% RSLogix 500 project fast_test.RSS, saved by version 8.30.00.16 %
PROJECT "UNTITLED"    % processor: Bul.1763 MicroLogix 1100 Series A %

PROGRAM FILES
  LAD 2 "MAIN"  6 rungs
  LAD 3 "CIRC_FIFO"  10 rungs

DATA FILES
  O0 OUTPUT  4 elements
  I1 INPUT  6 elements
  S2 STATUS  66 elements
  B3 BINARY  1 elements
  T4 TIMER  1 elements
  C5 COUNTER  1 elements
  R6 CONTROL  1 elements
  N7 INTEGER  6 elements
  F8 FLOAT  1 elements
  N252 LINE0  32 elements
  N253 LINE 1  32 elements
  N254 LINE 2  32 elements
  N255 LINE3  32 elements

LADDER 2 "MAIN"
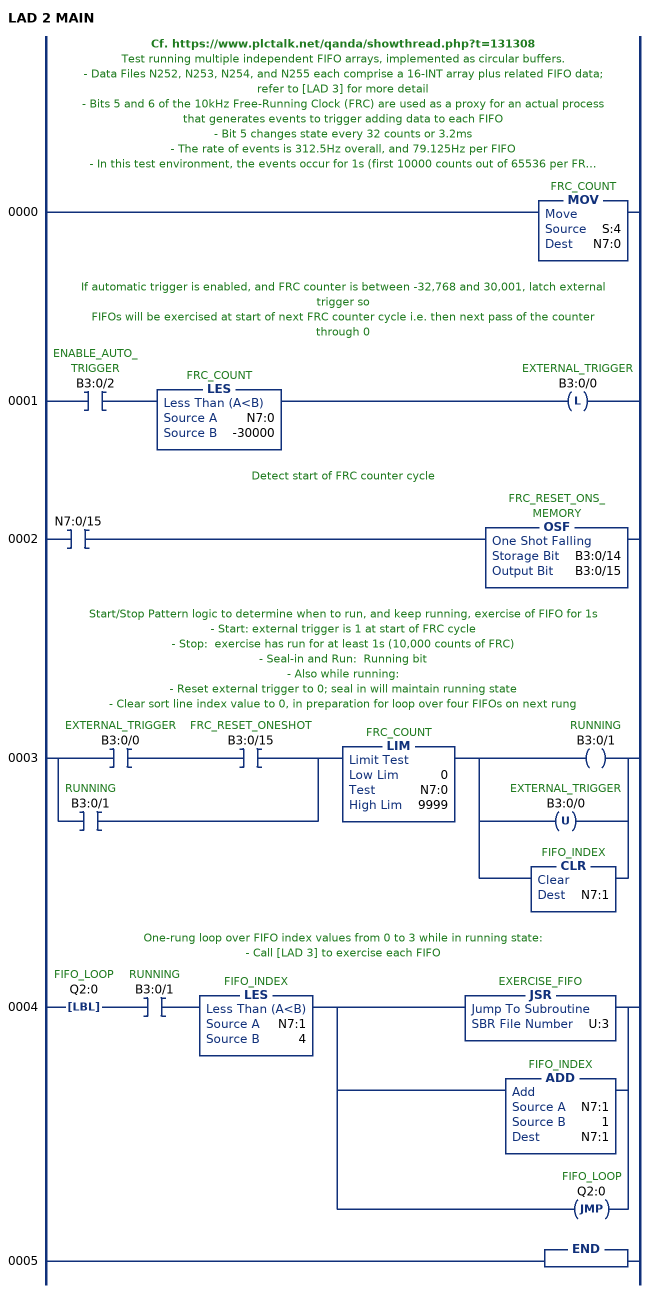
% Rung: 0 %
% TITLE: Cf. https://www.plctalk.net/qanda/showthread.php?t=131308 %
% Test running multiple independent FIFO arrays, implemented as circular buffers.
% - Data Files N252, N253, N254, and N255 each comprise a 16-INT array plus related FIFO data; refer to [LAD 3] for more detail
% - Bits 5 and 6 of the 10kHz Free-Running Clock (FRC) are used as a proxy for an actual process that generates events to trigger adding data to each FIFO
%   - Bit 5 changes state every 32 counts or 3.2ms
%   - The rate of events is 312.5Hz overall, and 79.125Hz per FIFO
% - In this test environment, the events occur for 1s (first 10000 counts out of 65536 per FRC cycle)
% - Events can be manually triggered for one cycle by assigning 1 as the value of the external trigger
%   - That external trigger value will be reset to 0 at the end of the cycle
% - Events can also be automatically and continuously triggered on every FRC cycle by manually assigning 1 to the automatic trigger
% 
% Rung 0000 - Copy current FRC counter value to local memory, so the value will not change throughout the scan
% Rung 0001 - Generate automatic trigger, if requested
% Rung 0002 - Detect start of FRC cycle
% Rung 0003 - Determine run state, i.e. when to exercise FIFOs
% Rung 0004 - While in running state, call subroutine (LAD 3] to exercise each FIFO %
SOR MOV S:4 N7:0 EOR
%   S:4  "Time Base" %
%   N7:0  FRC_COUNT %
% Rung: 1 %
% If automatic trigger is enabled, and FRC counter is between -32,768 and 30,001, latch external trigger so
% FIFOs will be exercised at start of next FRC counter cycle i.e. then next pass of the counter through 0 %
SOR XIC B3:0/2 LES N7:0 -30000 OTL B3:0/0 EOR
%   B3:0/2  ENABLE_AUTO_TRIGGER %
%   N7:0  FRC_COUNT %
%   B3:0/0  EXTERNAL_TRIGGER %
% Rung: 2 %
% Detect start of FRC counter cycle %
SOR XIC N7:0/15 OSF B3:0/14 B3:0/15 EOR
%   B3:0/14  FRC_RESET_ONS_MEMORY %
%   B3:0/15  FRC_RESET_ONESHOT %
% Rung: 3 %
% Start/Stop Pattern logic to determine when to run, and keep running, exercise of FIFO for 1s
% - Start: external trigger is 1 at start of FRC cycle
% - Stop:  exercise has run for at least 1s (10,000 counts of FRC)
% - Seal-in and Run:  Running bit
% - Also while running:
%   - Reset external trigger to 0; seal in will maintain running state
%   - Clear sort line index value to 0, in preparation for loop over four FIFOs on next rung %
SOR BST XIC B3:0/0 XIC B3:0/15 NXB XIC B3:0/1 BND LIM 0 N7:0 9999 BST OTE B3:0/1 NXB OTU B3:0/0 NXB CLR N7:1 BND EOR
%   B3:0/0  EXTERNAL_TRIGGER %
%   B3:0/15  FRC_RESET_ONESHOT %
%   B3:0/1  RUNNING %
%   N7:0  FRC_COUNT %
%   N7:1  FIFO_INDEX %
% Rung: 4 %
% One-rung loop over FIFO index values from 0 to 3 while in running state:
% - Call [LAD 3] to exercise each FIFO %
SOR LBL Q2:0 XIC B3:0/1 LES N7:1 4 BST JSR U:3 NXB ADD N7:1 1 N7:1 NXB JMP Q2:0 BND EOR
%   Q2:0  FIFO_LOOP %
%   B3:0/1  RUNNING %
%   N7:1  FIFO_INDEX %
%   U:3  EXERCISE_FIFO %
% Rung: 5 %
SOR END EOR

LADDER 3 "CIRC_FIFO"
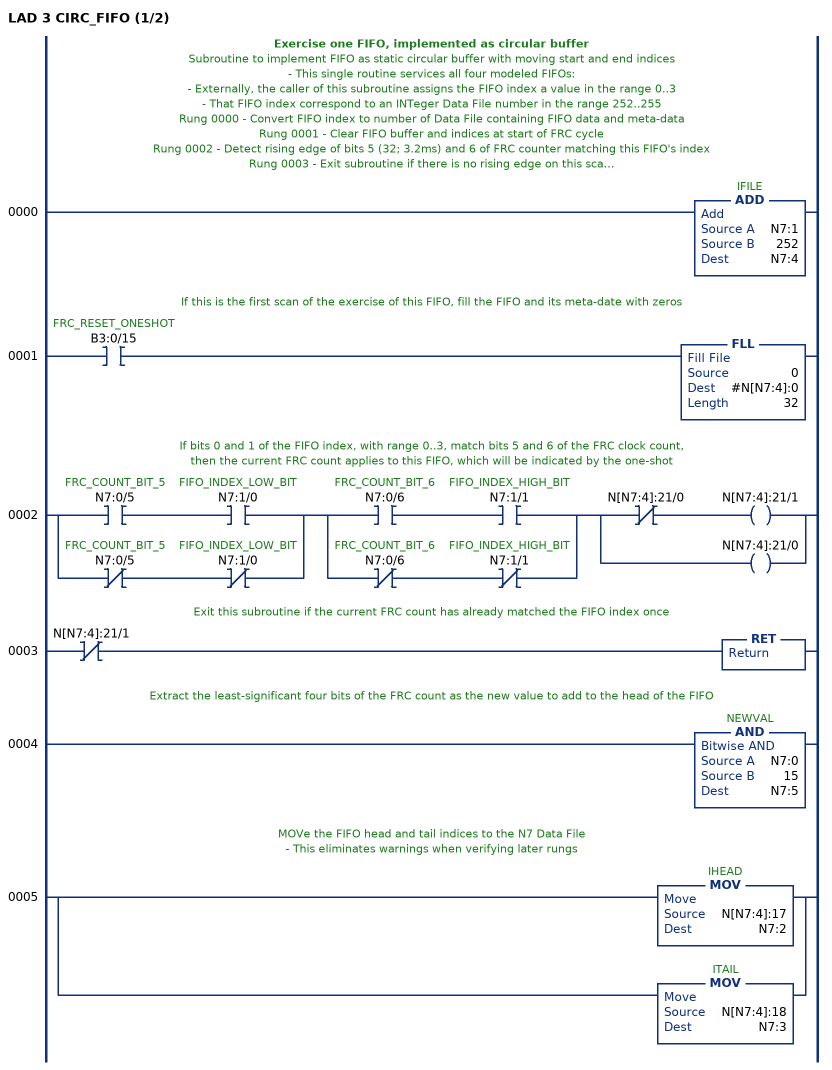
% Rung: 0 %
% TITLE: Exercise one FIFO, implemented as circular buffer %
% Subroutine to implement FIFO as static circular buffer with moving start and end indices
% - This single routine services all four modeled FIFOs:
%   - Externally, the caller of this subroutine assigns the FIFO index a value in the range 0..3
%   - That FIFO index correspond to an INTeger Data File number in the range 252..255
% 
% Rung 0000 - Convert FIFO index to number of Data File containing FIFO data and meta-data
% Rung 0001 - Clear FIFO buffer and indices at start of FRC cycle
% Rung 0002 - Detect rising edge of bits 5 (32; 3.2ms) and 6 of FRC counter matching this FIFO's index
% Rung 0003 - Exit subroutine if there is no rising edge on this scan
% Rung 0004 - Calculate new value to push onto FIFO
% Rung 0005 - Copy head and tail indices from this FIFO's file
% Rung 0006 - If circular buffer is full, then unload FIFO tail value and increment FIFO tail index
% Rung 0007 - load FIFO head value and increment FIFO head index
% Rung 0008 - Increment number of values added to FIFO
% 
% The four Data Files contain the FIFOS are N252, N253, N254, and N255, plus FIFO-related meta-data.
% The Data Files are referred to here as N[N7:4], where N7:4 is the file number (252..255), which is the FIFO index (N7:1) with a range of 0..3 plus 252
% Each file comprises
% - :0..:15 - A 16-element circular buffer
% - :[N7:3] - The head (new) element
% - :[N7:3] - The tail (oldest) element
% - :16 - The running count of items loaded into the head of the buffer
% - :17 - The head index, where the next new value will be added; :17's head index value will be MOVed to N7:3, then incremented and put back into :17
% - :18 - The tail index, where the oldest value is; if used, then :18's value will be MOVed to N7:2, the incremented an put back into :18
% - :19 - The new value to be loaded (not used); this will be
% - :20 - The oldest value that has been unloaded
% - :21 - Bits used by the FIFO
% - :21/0 - Memory for the one-shot
% - :21/1 - The one-shot itself, which detects the first scan when the FRC count bits 5 and 6 match the FIFO number %
SOR ADD N7:1 252 N7:4 EOR
%   N7:1  FIFO_INDEX %
%   N7:4  IFILE %
% Rung: 1 %
% If this is the first scan of the exercise of this FIFO, fill the FIFO and its meta-date with zeros %
SOR XIC B3:0/15 FLL 0 #N[N7:4]:0 32 EOR
%   B3:0/15  FRC_RESET_ONESHOT %
%   N7:4  IFILE %
% Rung: 2 %
% If bits 0 and 1 of the FIFO index, with range 0..3, match bits 5 and 6 of the FRC clock count,
% then the current FRC count applies to this FIFO, which will be indicated by the one-shot %
SOR BST XIC N7:0/5 XIC N7:1/0 NXB XIO N7:0/5 XIO N7:1/0 BND BST XIC N7:0/6 XIC N7:1/1 NXB XIO N7:0/6 XIO N7:1/1 BND BST XIO N[N7:4]:21/0 OTE N[N7:4]:21/1 NXB OTE N[N7:4]:21/0 BND EOR
%   N7:0/5  FRC_COUNT_BIT_5 %
%   N7:1/0  FIFO_INDEX_LOW_BIT %
%   N7:0/6  FRC_COUNT_BIT_6 %
%   N7:1/1  FIFO_INDEX_HIGH_BIT %
%   N7:4  IFILE %
% Rung: 3 %
% Exit this subroutine if the current FRC count has already matched the FIFO index once %
SOR XIO N[N7:4]:21/1 RET EOR
%   N7:4  IFILE %
% Rung: 4 %
% Extract the least-significant four bits of the FRC count as the new value to add to the head of the FIFO %
SOR AND N7:0 15 N7:5 EOR
%   N7:0  FRC_COUNT %
%   N7:5  NEWVAL %
% Rung: 5 %
% MOVe the FIFO head and tail indices to the N7 Data File
% - This eliminates warnings when verifying later rungs %
SOR BST MOV N[N7:4]:17 N7:2 NXB MOV N[N7:4]:18 N7:3 BND EOR
%   N7:4  IFILE %
%   N7:2  IHEAD %
%   N7:3  ITAIL %

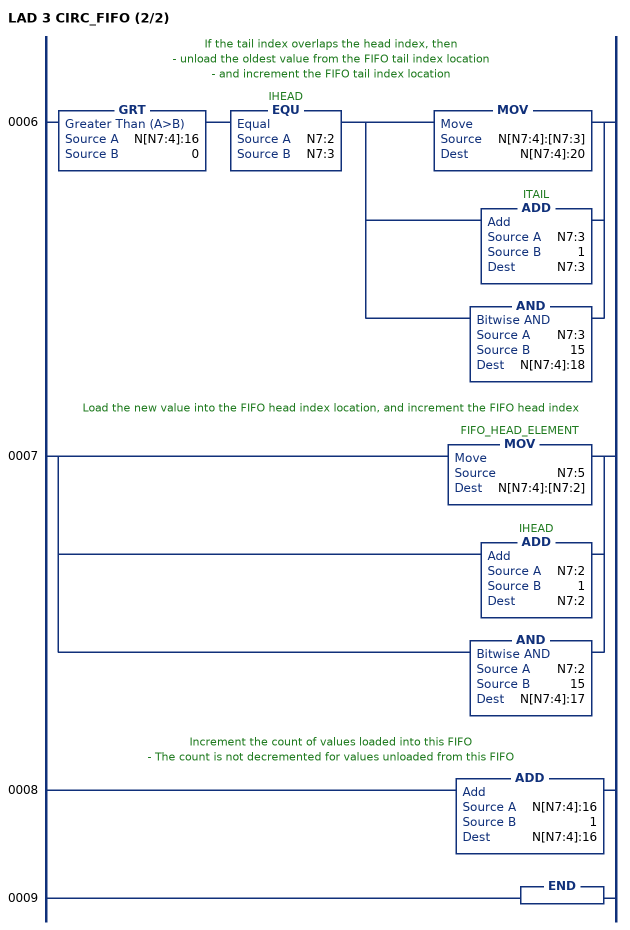
% Rung: 6 %
% If the tail index overlaps the head index, then
% - unload the oldest value from the FIFO tail index location
% - and increment the FIFO tail index location %
SOR GRT N[N7:4]:16 0 EQU N7:2 N7:3 BST MOV N[N7:4]:[N7:3] N[N7:4]:20 NXB ADD N7:3 1 N7:3 NXB AND N7:3 15 N[N7:4]:18 BND EOR
%   N7:4  IFILE %
%   N7:2  IHEAD %
%   N7:3  ITAIL %
%   N[N7:4]:[N7:3]  FIFO_TAIL_ELEMENT %
% Rung: 7 %
% Load the new value into the FIFO head index location, and increment the FIFO head index %
SOR BST MOV N7:5 N[N7:4]:[N7:2] NXB ADD N7:2 1 N7:2 NXB AND N7:2 15 N[N7:4]:17 BND EOR
%   N7:5  NEWVAL %
%   N[N7:4]:[N7:2]  FIFO_HEAD_ELEMENT %
%   N7:4  IFILE %
%   N7:2  IHEAD %
% Rung: 8 %
% Increment the count of values loaded into this FIFO
% - The count is not decremented for values unloaded from this FIFO %
SOR ADD N[N7:4]:16 1 N[N7:4]:16 EOR
%   N7:4  IFILE %
% Rung: 9 %
SOR END EOR

OTHER DOCUMENTED ADDRESSES
  C5:0.ACC  1DS_INTERVAL_COUNT
  N[N7:4]:000  CIRCULAR_BUFFER
  N[N7:4]:016  FIFO_COUNT
  N[N7:4]:017  FIFO_HEAD
  N[N7:4]:018  FIFO_TAIL
  N[N7:4]:019  FIFO_NEWVAL
  N[N7:4]:020  FIFO_OLDVAL
  N[N7:4]:021  FIFO_BITS
  N[N7:4]:021/00  FIFO_ONESHOT_MEMORY
  N[N7:4]:021/01  FIFO_ONESHOT

COMMENTS NOT ATTACHED TO A CURRENT RUNG
  N7:0: Cf. https://www.plctalk.net/qanda/showthread.php?t=131308

DATA TABLE (non-zero values as saved)
DATA R6
% .LEN .POS %
% R6:0 % 128 0
DATA N7
% N7:0 % 0 0 0 0 252 0
